FUNCTION_BLOCK INTERNAL Fb_EdgeDetector
VAR_INPUT
	inputValue		: BOOL;
END_VAR
VAR_OUTPUT
	risingEdge		: BOOL;
	fallingEdge		: BOOL;
END_VAR
VAR
	lastValue 		: BOOL;
	tlastPush		: TIME := TIME();  // initialize with now
	tDelayValue     : TIME := T#10MS;
END_VAR

// if a change happened and new values get accepted
IF(inputValue <> lastValue AND (tlastPush + tDelayValue) < TIME()) THEN
	IF(inputValue) THEN
		risingEdge := TRUE;
		fallingEdge := FALSE;
	ELSE
		risingEdge := FALSE;
		fallingEdge := TRUE;
	END_IF
	lastValue := inputValue;  // overwrite stored value
	tlastPush := TIME();
END_IF

END_FUNCTION_BLOCK

(* stored: Version 1.1.0.1, ProductVersion 3.1.4024.9
   POU Fb_EdgeDetector: Id {d746b410-be40-4fa8-9299-53feae6bfcc6}, SpecialFunc None *)
